GLOBALCONSTANTS DefaultPool_Bargraph (* Bargraph geometry and scale constants (Length, ScalePx, Min, Max, Type) *)
  PACKAGE Uebungen::const::UT::HystereseHorizontal;
  VAR_GLOBAL CONSTANT
    Bargraph_Hysterese_ScalePx : REAL := 1.86;
    Bargraph_Hysterese_LengthPx : REAL := 186.0;
    Bargraph_Hysterese_Min : REAL := 0.0;
    Bargraph_Hysterese_Max : REAL := 100.0;
    Bargraph_Hysterese_Type : USINT := 3;
  END_VAR
END_GLOBALCONSTANTS
